// TIA Portal V16 export
// export: Created 2022-01-12T14:32:03.9624873Z, ExportSetting WithDefaults, DisplayName Totally Integrated Automation Portal, DisplayVersion V16 Update 4, DisplayName TIA Portal Version Control Interface, DisplayVersion V16 Update 2, DisplayName TIA Portal Openness, DisplayVersion V16 Update 4, DisplayName STEP 7 Professional, DisplayVersion V16 Update 4, DisplayName STEP 7 Safety, DisplayVersion V16, DisplayName WinCC Professional, DisplayVersion V16 Update 4
DATA_BLOCK "ms_na_procenty_DB"   // DB34
{ S7_Optimized_Access := 'TRUE' }
VERSION : 0.1
// blok danych dla funkcji ms_na_procenty
// stored: AutoNumber true, DBAccessibleFromOPCUA true, IsOnlyStoredInLoadMemory false, IsRetainMemResEnabled false, IsWriteProtectedInAS false, MemoryReserve 100
   VAR RETAIN
      inJednostkaAlkaliczna : Real;   // 1% środka alkalicznego= 48mS
      inJednostkaKwaśna : Real;   // 1% środka kwaśnego=56mS
      inPrzewodnośćCzystejWody { S7_SetPoint := 'True'} : Real;   // Przewodność czystej wody=0.3mS
   END_VAR
   VAR
      outStężenieŚrodkaTor1 : Real;
      outStężenieŚrodkaTor2 : Real;
   END_VAR
BEGIN
END_DATA_BLOCK
